// TIA Portal V17 export
// export: Created 2024-03-30T11:14:40.7482284Z, ExportSetting WithDefaults, DisplayName Totally Integrated Automation Portal, DisplayVersion V17, DisplayName TIA Portal Openness, DisplayVersion V17, DisplayName TIA Portal Version Control Interface, DisplayVersion V17, DisplayName STEP 7 Professional, DisplayVersion V17, DisplayName STEP 7 Safety, DisplayVersion V17, DisplayName WinCC Advanced, DisplayVersion V17
DATA_BLOCK "PRG_VGR_Axis_horizontal_DB"   // DB8
AUTHOR : A.Schaefer
VERSION : 0.1
// stored: AutoNumber true, DBAccessibleFromOPCUA true, DBAccessibleFromWebserver true, InstanceOfName PRG_VGR_Axis_horizontal, InstanceOfType FB
"PRG_VGR_Axis_horizontal"
   // VAR
   //    lx_Init { ExternalAccessible := 'False'; ExternalVisible := 'False'; ExternalWritable := 'False'} : Bool;
   //    lfb_horizontal_Axis { ExternalAccessible := 'False'; ExternalVisible := 'False'; ExternalWritable := 'False'} : "FB_Axis_Auto";
   // END_VAR
BEGIN
END_DATA_BLOCK
